TEXTLIST TextList_AccessLevel
  0 = 'GUEST'
  1 = 'OPERATOR'
  2 = 'TECHNICIAN'
  3 = 'ENGINEER'
  4 = 'MANAGER'
  5 = 'JKS'
   = ''
END_TEXTLIST

(* stored: Version 1.1.0.1, ProductVersion 3.1.4024.12
   TextList TextList_AccessLevel: Id {5240aac9-530b-40f6-be71-0583f7df25f7} *)
